{attribute addProperty BoxType "EL1002--0000"}
{attribute addProperty Id "ChannelAT %I*ARRAY[0..1] OF Channel_E4AEF59E1620WcStateAT %I*WcState_98A4DF7520.250InfoDataAT %I*InfoData_192954DE1620"}
{attribute addProperty CRC "672950472"}
{attribute addProperty SizeInBites "34"}
{attribute addProperty SizeInBytes "4.25"}
TYPE EL1002_37B2B160 :
STRUCT
	{attribute addProperty Name "Channel"}
	Channel : ARRAY[0..1] OF Channel_E4AEF59E;
	{attribute addProperty Name "WcState"}
	WcState : WcState_98A4DF75;
	{attribute addProperty Name "InfoData"}
	InfoData : InfoData_192954DE;
END_STRUCT
END_TYPE

(* stored: Version 1.2.0.0, ProductVersion 3.1.4024.9
   DUT EL1002_37B2B160: Id {b4d6432a-1492-48f2-9876-8cdb48ef5e7d} *)
